// TIA Portal V20 export
DATA_BLOCK "GLOBAL_GRAPH_HMI_IF_DB"   // DB205
{ S7_Optimized_Access := 'TRUE' }
// stored: AutoNumber false, MemoryReserve 100
   VAR
      GRAPH : Array[0..10] of "GRAPH_CONTROL_UDT";
   END_VAR
BEGIN
   // GRAPH[1] : ST010_MAIN_GRAPH_FB
   // GRAPH[2] : ST020_CNV06_GRAPH_FB
   // GRAPH[3] : ST020_CNV04_GRAPH_FB
   // GRAPH[4] : ST020_CNV05_GRAPH_FB
   // GRAPH[5] : ST020_MAIN_GRAPH_FB
   // GRAPH[6] : ST020_ROBOT_GRAPH_FB
   // GRAPH[7] : ST020_RB01_GRAPH_FB
   // GRAPH[8] : ST020_RB02_GRAPH_FB
   // GRAPH[9] : ST020_RB06_GRAPH_FB
   // GRAPH[10] : ST025_RB01_GRAPH_FB
END_DATA_BLOCK
